// Mitsubishi GX Works2 project: Group22 temp   PLC: FX3G

// global labels: Global1
VAR_GLOBAL
  startMachine AT X010 : BOOL;  (* start machine 1 bottom *)
  machineON AT M0 : BOOL;  (* indication for machine 1 is on *)
  senTouch AT X001 : BOOL;  (* is on if the sensor for the machine sense a tray to execute ziluf *)
  sen_30 AT X003 : BOOL;  (* indication for lower temperature then 30 *)
  sen_15 AT X002 : BOOL;  (* indication for lower temperature then 15 *)
  startDay AT X007 : BOOL;  (* start day bottom *)
  creamInput AT D1119 : REAL;  (* input for cream inventory *)
  creamQuantity AT D1121 : REAL;  (* current quantity of cream in the inventory *)
  chocolateInput AT D1123 : REAL;  (* input for chocolate inventory *)
  chocolateQuantity AT D1125 : REAL;  (* chocolate current quantity *)
  biscuitInput AT D1127 : REAL;  (* input for biscuit inventory *)
  biscuitQuantity AT D1129 : REAL;  (* biscuit current quantity *)
END_VAR
VAR_GLOBAL CONSTANT
  minCream : REAL := 300;  (* minimum quantity needed of cream *)
  minChocolate : REAL := 240;  (* minimum quantity needed of chocolate *)
  minBiscuit : REAL := 6;  (* minimum quantity needed of biscuite *)
END_VAR
VAR_GLOBAL
  notAllQuantitiesGood AT M1 : BOOL;  (* is on if NOT all input quantities are enough for starting the day *)
  counter3sec AT TC1 : BOOL;  (* counter for the y7 blinks at the end of the day *)
END_VAR
VAR_GLOBAL CONSTANT
  fullTime : INT := 30;  (* time of blinking y7 at end day *)
END_VAR
VAR_GLOBAL
  stopAfter3Sec AT TS1 : BOOL;  (* counter for stop blinking of Y7 after 3 seconds *)
  timerReset AT M3 : BOOL;  (* rest timer for counter 5 units packed *)
  timer1 AT TC2 : BOOL;  (* timer name for blinking time of M4 *)
END_VAR
VAR_GLOBAL CONSTANT
  timeInterval : INT := 5;  (* time interval for light on while blinking *)
END_VAR
VAR_GLOBAL
  endTimer1 AT TS2 : BOOL;  (* end timer for blinking fictive light *)
  timer2 AT TC3 : BOOL;  (* timer name for blinking time of M5 *)
  endTimer2 AT TS3 : BOOL;  (* end timer for blinking fictive light that represents Y7 *)
  productionLight AT Y007 : BOOL;  (* light that works all day *)
  fictiveBlinkLight1 AT M4 : BOOL;  (* fictive light that blinks together with Y7 to stimulate Y7 blinks *)
  fictiveBlinkLight2 AT M5 : BOOL;  (* fictive light that represents Y7 *)
  fictiveProductionLight AT M6 : BOOL;  (* production day - process is currently happening *)
  startZilof AT X011 : BOOL;  (* transfer cream from inventory to containter to start zilof stage *)
END_VAR
VAR_GLOBAL CONSTANT
  creamToUse : REAL := 300;  (* amount of cream to use in 1 iteration *)
  biscuitToUse : REAL := 6;  (* amount of bixcuit to use in 1 iteration *)
END_VAR
VAR_GLOBAL
  zilofContainer AT D1131 : REAL;  (* current quantity of cream in the container *)
  counter4seC AT TS4 : BOOL;  (* counter time to blink while transfering *)
END_VAR
VAR_GLOBAL CONSTANT
  blinkTime : INT := 40;  (* time of blinking y0 and y1 at transport from zilof stage to dipping stage *)
END_VAR
VAR_GLOBAL
  timerReset2 AT M7 : BOOL;  (* reset timer for counter of last unit to pack *)
  timer3 AT TC5 : BOOL;  (* timer name for blinking time of Y0 *)
  endTimer3 AT TS5 : BOOL;  (* end timer for blinking Y0 *)
  lightBlink1 AT Y000 : BOOL;  (* blinkig light Y0 to moving units form ziluf *)
  timer4 AT TC6 : BOOL;  (* timer name for blinking time of Y1 *)
  lightBlink2 AT Y001 : BOOL;  (* blinkig light Y1 to moving units form ziluf *)
  endTimer4 AT TS6 : BOOL;  (* end timer for blinking Y1 *)
  zilufON AT Y004 : BOOL;  (* light that stay on while we are in zilof stage *)
  cam AT X004 : BOOL;  (* indication for finish zilof stage *)
  dipInChocolate AT X006 : BOOL;  (* sample the analog input 1 *)
  dipTimer AT TC7 : BOOL;  (* timer for the dipping stage *)
END_VAR
VAR_GLOBAL CONSTANT
  dipInterval : INT := 50;  (* duration time to dip in chocolate *)
END_VAR
VAR_GLOBAL
  dipStop AT TS7 : BOOL;  (* after 5 seconds Y3 sets off *)
  dipInChocolateOn AT Y003 : BOOL;  (* indication for dip process *)
  afterZiluf AT M8 : BOOL;  (* the tray is out of machine a, finished zilufh *)
  iterationDone AT M100 : BOOL;  (* full iteration tray production is done *)
  finishtransferBlink AT M9 : BOOL;  (* after blinking for 4 seconds, turns on *)
  shutDown AT X005 : BOOL;  (* emergency bottom *)
  sampleValue AT D8201 : INT;  (* sample value from anaolog input 1 *)
END_VAR
VAR_GLOBAL CONSTANT
  normalizationFactor : INT := 400;  (* factor to make analog input value shown as the screen *)
END_VAR
VAR_GLOBAL
  finishSampleAnalog AT M10 : BOOL;  (* done sampaling from analog 1 *)
  analog_input_1 AT D8280 : INT;  (* analog input 1 value *)
END_VAR
VAR_GLOBAL CONSTANT
  maxNormalDip : INT := 6;  (* if sample is less than 6 then normal dip *)
END_VAR
VAR_GLOBAL
  normalChocolateDip AT M11 : BOOL;  (* normal chocolate needed *)
  doubledChocolateDip AT M12 : BOOL;  (* double chocolate dip needed *)
END_VAR
VAR_GLOBAL CONSTANT
  amountDoubledDip : REAL := 240;  (* amount of chocolate to coat a tray with doubled amount *)
  amountNormalDip : REAL := 120;  (* amount of chocolate to coat a tray with normal amount *)
END_VAR
VAR_GLOBAL
  coatContainer AT D1135 : REAL;  (* container for coating chocolate above kremboes *)
  finishFillCoatContainer AT M13 : BOOL;  (* indication of end dipping stage *)
  packCounter AT CC1 : BOOL;  (* counter for how much krembo we pack in single iteration *)
END_VAR
VAR_GLOBAL CONSTANT
  packCounterValueLast : INT := 5;  (* number of krembos before the last one *)
END_VAR
VAR_GLOBAL
  packunit AT X000 : BOOL;  (* if on, a krembo unit is getting packed *)
  finishCoating AT M14 : BOOL;  (* if coating process is finished and Y3 turns off *)
  lastPackNeededOn AT Y002 : BOOL;  (* is on if only one last unit left to pack *)
  outCC1 AT CS1 : BOOL;  (* output of counter for 5 unit packs *)
  lastPackCounter AT CC2 : BOOL;  (* counter name of counter for last unit packing *)
END_VAR
VAR_GLOBAL CONSTANT
  packCounterValueLastuUnit : INT := 2;  (* counter for the last unit needed to be packed *)
END_VAR
VAR_GLOBAL
  outCC2 AT CS2 : BOOL;  (* output of counter for last unit pack *)
  readyKrembo AT D2015 : INT;  (* the ready krembos *)
END_VAR
VAR_GLOBAL CONSTANT
  magashKrembo : INT := 6;  (* number of krembos in one iteration *)
END_VAR
VAR_GLOBAL
  kremboOutput AT D8282 : INT;  (* output for the number o ready krembos in tens *)
END_VAR
VAR_GLOBAL CONSTANT
  normalizationFactor2 : INT := 40;  (* factor to make analog input value shown as the screen *)
END_VAR
VAR_GLOBAL
  enoughCreamInContainer AT M15 : BOOL;  (* indication of enough cream in the container to start zilof stage *)
  afterMovingToZilufContainer AT M20 : BOOL;  (* help light to indicate that we are after moving to ziluf container *)
END_VAR

// task Task_01 (event TRUE, interval 0, priority 31): POU_01

PROGRAM POU_01
(* structured ladder/FBD written out as ST: instructions are called as NAME(EN, inputs, outputs); _pN, _eN, _tN stand for wires *)
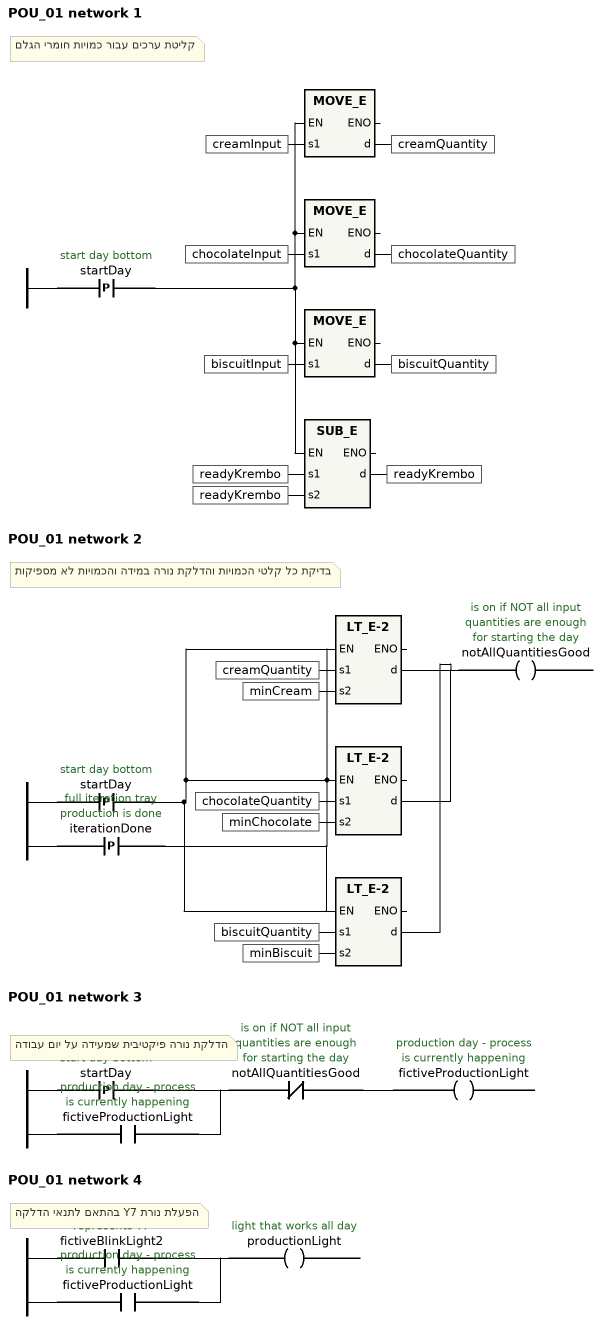
(* network 1 *)
(* קליטת ערכים עבור כמויות חומרי הגלם *)
_p1 := LDP(TRUE, startDay);
MOVE_E(_p1, creamInput, creamQuantity);
MOVE_E(_p1, chocolateInput, chocolateQuantity);
MOVE_E(_p1, biscuitInput, biscuitQuantity);
SUB_E(_p1, readyKrembo, readyKrembo, readyKrembo);
(* network 2 *)
(* בדיקת כל קלטי הכמויות והדלקת נורה במידה והכמויות לא מספיקות *)
_p1 := LDP(TRUE, startDay) OR LDP(TRUE, iterationDone);
LT_E(_p1, creamQuantity, minCream, _t2);
LT_E(_p1, chocolateQuantity, minChocolate, _t3);
LT_E(_p1, biscuitQuantity, minBiscuit, _t4);
notAllQuantitiesGood := _t2 OR _t3 OR _t4;
(* network 3 *)
(* הדלקת נורה פיקטיבית שמעידה על יום עבודה *)
fictiveProductionLight := (LDP(TRUE, startDay) OR fictiveProductionLight) AND NOT notAllQuantitiesGood;
(* network 4 *)
(* הפעלת נורת Y7 בהתאם לתנאי הדלקה *)
productionLight := fictiveBlinkLight2 OR fictiveProductionLight;
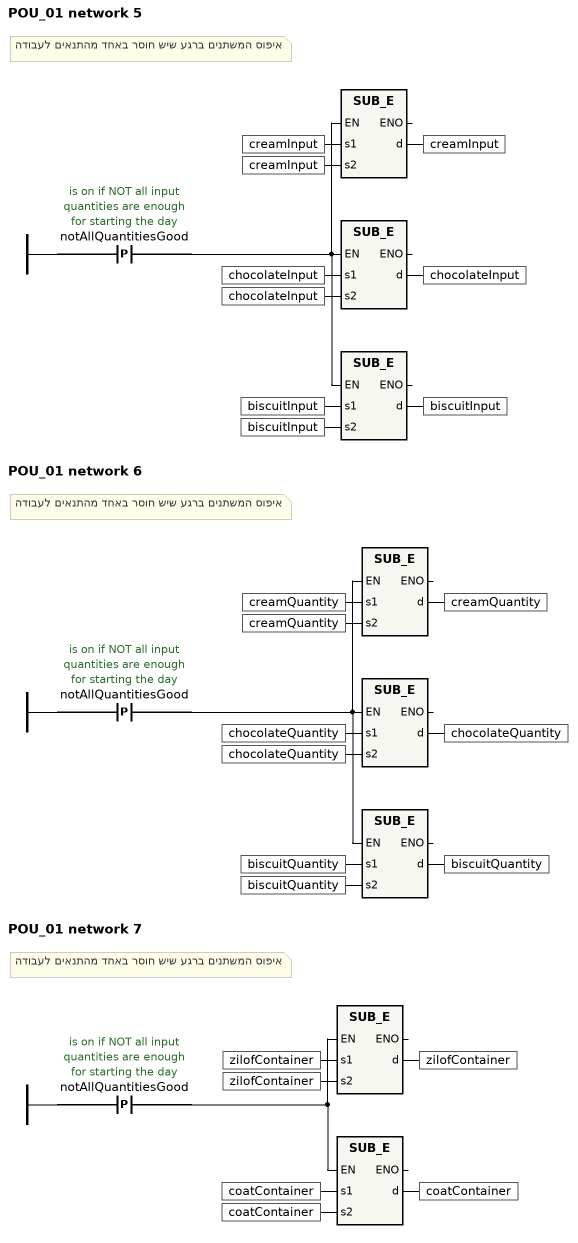
(* network 5 *)
(* איפוס המשתנים ברגע שיש חוסר באחד מהתנאים לעבודה *)
_p1 := LDP(TRUE, notAllQuantitiesGood);
SUB_E(_p1, creamInput, creamInput, creamInput);
SUB_E(_p1, chocolateInput, chocolateInput, chocolateInput);
SUB_E(_p1, biscuitInput, biscuitInput, biscuitInput);
(* network 6 *)
(* איפוס המשתנים ברגע שיש חוסר באחד מהתנאים לעבודה *)
_p1 := LDP(TRUE, notAllQuantitiesGood);
SUB_E(_p1, creamQuantity, creamQuantity, creamQuantity);
SUB_E(_p1, chocolateQuantity, chocolateQuantity, chocolateQuantity);
SUB_E(_p1, biscuitQuantity, biscuitQuantity, biscuitQuantity);
(* network 7 *)
(* איפוס המשתנים ברגע שיש חוסר באחד מהתנאים לעבודה *)
_p1 := LDP(TRUE, notAllQuantitiesGood);
SUB_E(_p1, zilofContainer, zilofContainer, zilofContainer);
SUB_E(_p1, coatContainer, coatContainer, coatContainer);
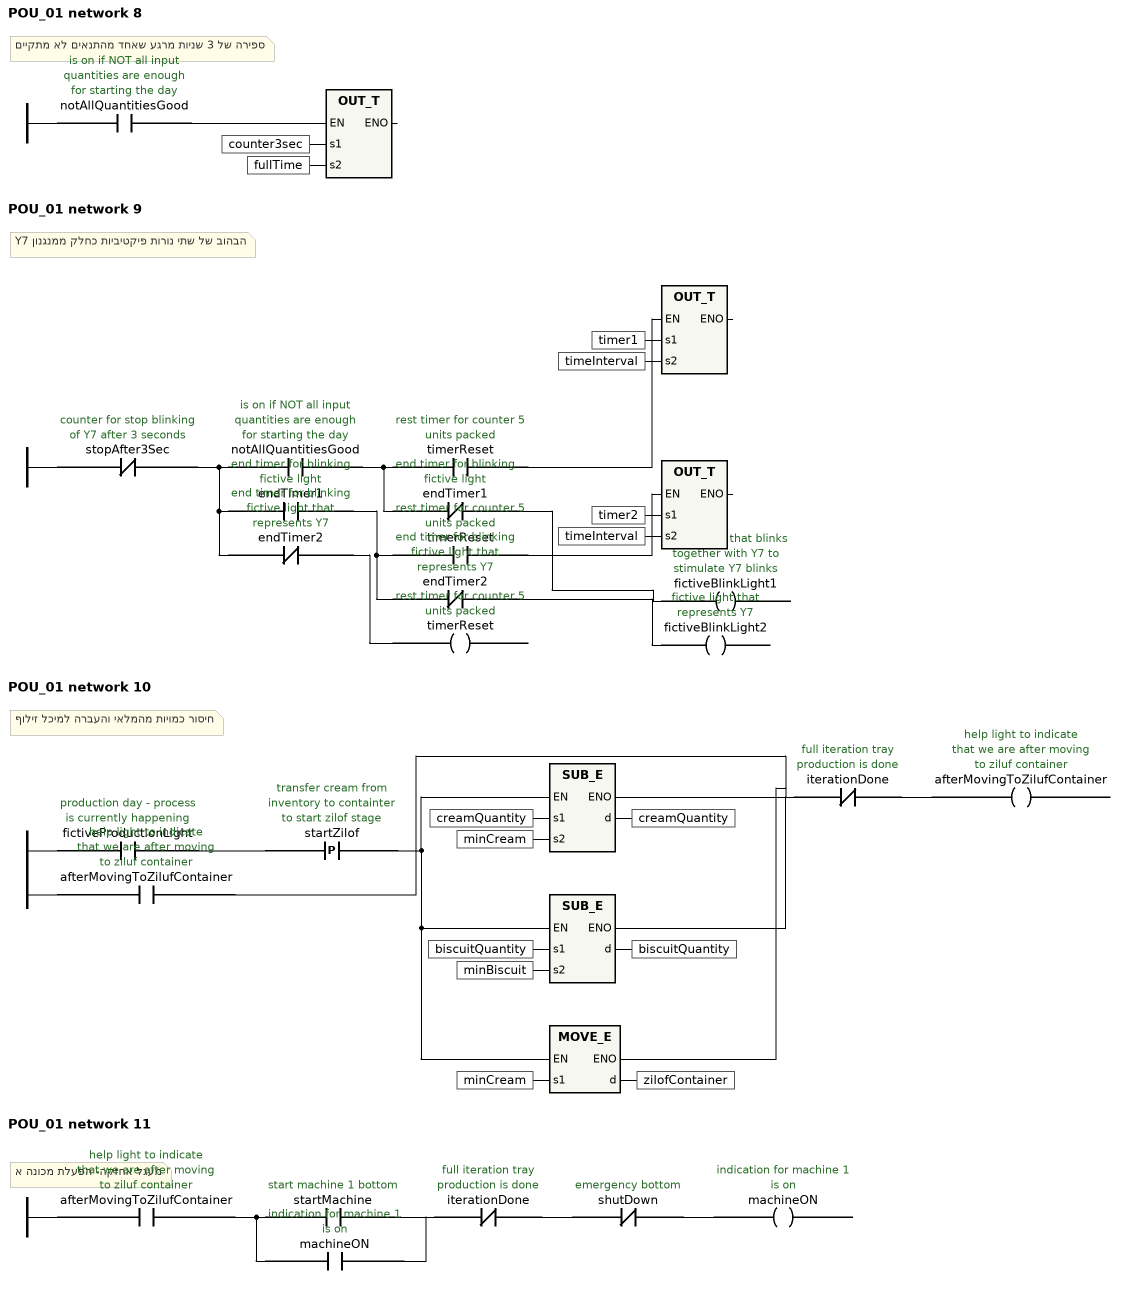
(* network 8 *)
(* ספירה של 3 שניות מרגע שאחד מהתנאים לא מתקיים *)
OUT_T(notAllQuantitiesGood, counter3sec, fullTime);
(* network 9 *)
(* הבהוב של שתי נורות פיקטיביות כחלק ממנגנון Y7 *)
_p1 := NOT stopAfter3Sec;
_p2 := _p1 AND notAllQuantitiesGood;
OUT_T(_p2 AND timerReset, timer1, timeInterval);
fictiveBlinkLight1 := _p2 AND NOT endTimer1;
_p3 := _p1 AND endTimer1;
OUT_T(_p3 AND timerReset, timer2, timeInterval);
fictiveBlinkLight2 := _p3 AND NOT endTimer2;
timerReset := _p1 AND NOT endTimer2;
(* network 10 *)
(* חיסור כמויות מהמלאי והעברה למיכל זילוף *)
_p1 := fictiveProductionLight AND LDP(TRUE, startZilof);
_e2 := SUB_E(_p1, creamQuantity, minCream, creamQuantity);
_e3 := SUB_E(_p1, biscuitQuantity, minBiscuit, biscuitQuantity);
_e4 := MOVE_E(_p1, minCream, zilofContainer);
afterMovingToZilufContainer := (_e2 OR _e3 OR _e4 OR afterMovingToZilufContainer) AND NOT iterationDone;
(* network 11 *)
(* מעגל אחזקה- הפעלת מכונה א *)
machineON := (((afterMovingToZilufContainer AND startMachine) OR (afterMovingToZilufContainer AND machineON)) AND NOT iterationDone) AND NOT shutDown;
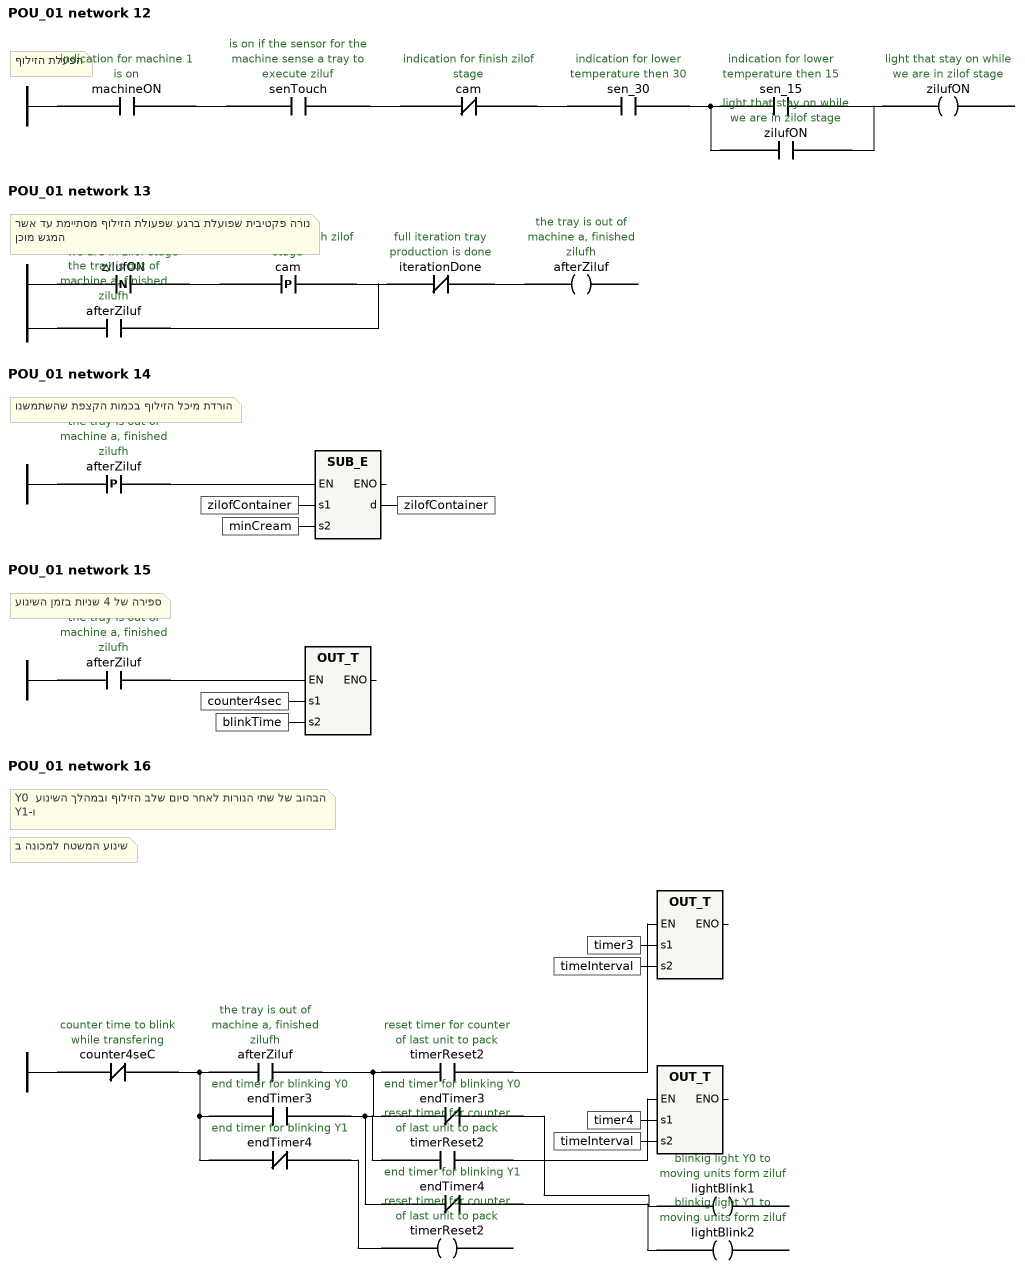
(* network 12 *)
(* הפעלת הזילוף *)
_p1 := machineON AND senTouch AND NOT cam AND sen_30;
zilufON := (_p1 AND sen_15) OR (_p1 AND zilufON);
(* network 13 *)
(* נורה פקטיבית שפועלת ברגע שפעולת הזילוף מסתיימת עד אשר המגש מוכן *)
afterZiluf := ((LDF(TRUE, zilufON) AND LDP(TRUE, cam)) OR afterZiluf) AND NOT iterationDone;
(* network 14 *)
(* הורדת מיכל הזילוף בכמות הקצפת שהשתמשנו *)
SUB_E(LDP(TRUE, afterZiluf), zilofContainer, minCream, zilofContainer);
(* network 15 *)
(* ספירה של 4 שניות בזמן השינוע *)
OUT_T(afterZiluf, counter4sec, blinkTime);
(* network 16 *)
(* הבהוב של שתי הנורות לאחר סיום שלב הזילוף ובמהלך השינוע  Y0 ו-Y1 *)
(* שינוע המשטח למכונה ב *)
_p1 := NOT counter4seC;
_p2 := _p1 AND afterZiluf;
OUT_T(_p2 AND timerReset2, timer3, timeInterval);
lightBlink1 := _p2 AND NOT endTimer3;
_p3 := _p1 AND endTimer3;
OUT_T(_p3 AND timerReset2, timer4, timeInterval);
lightBlink2 := _p3 AND NOT endTimer4;
timerReset2 := _p1 AND NOT endTimer4;
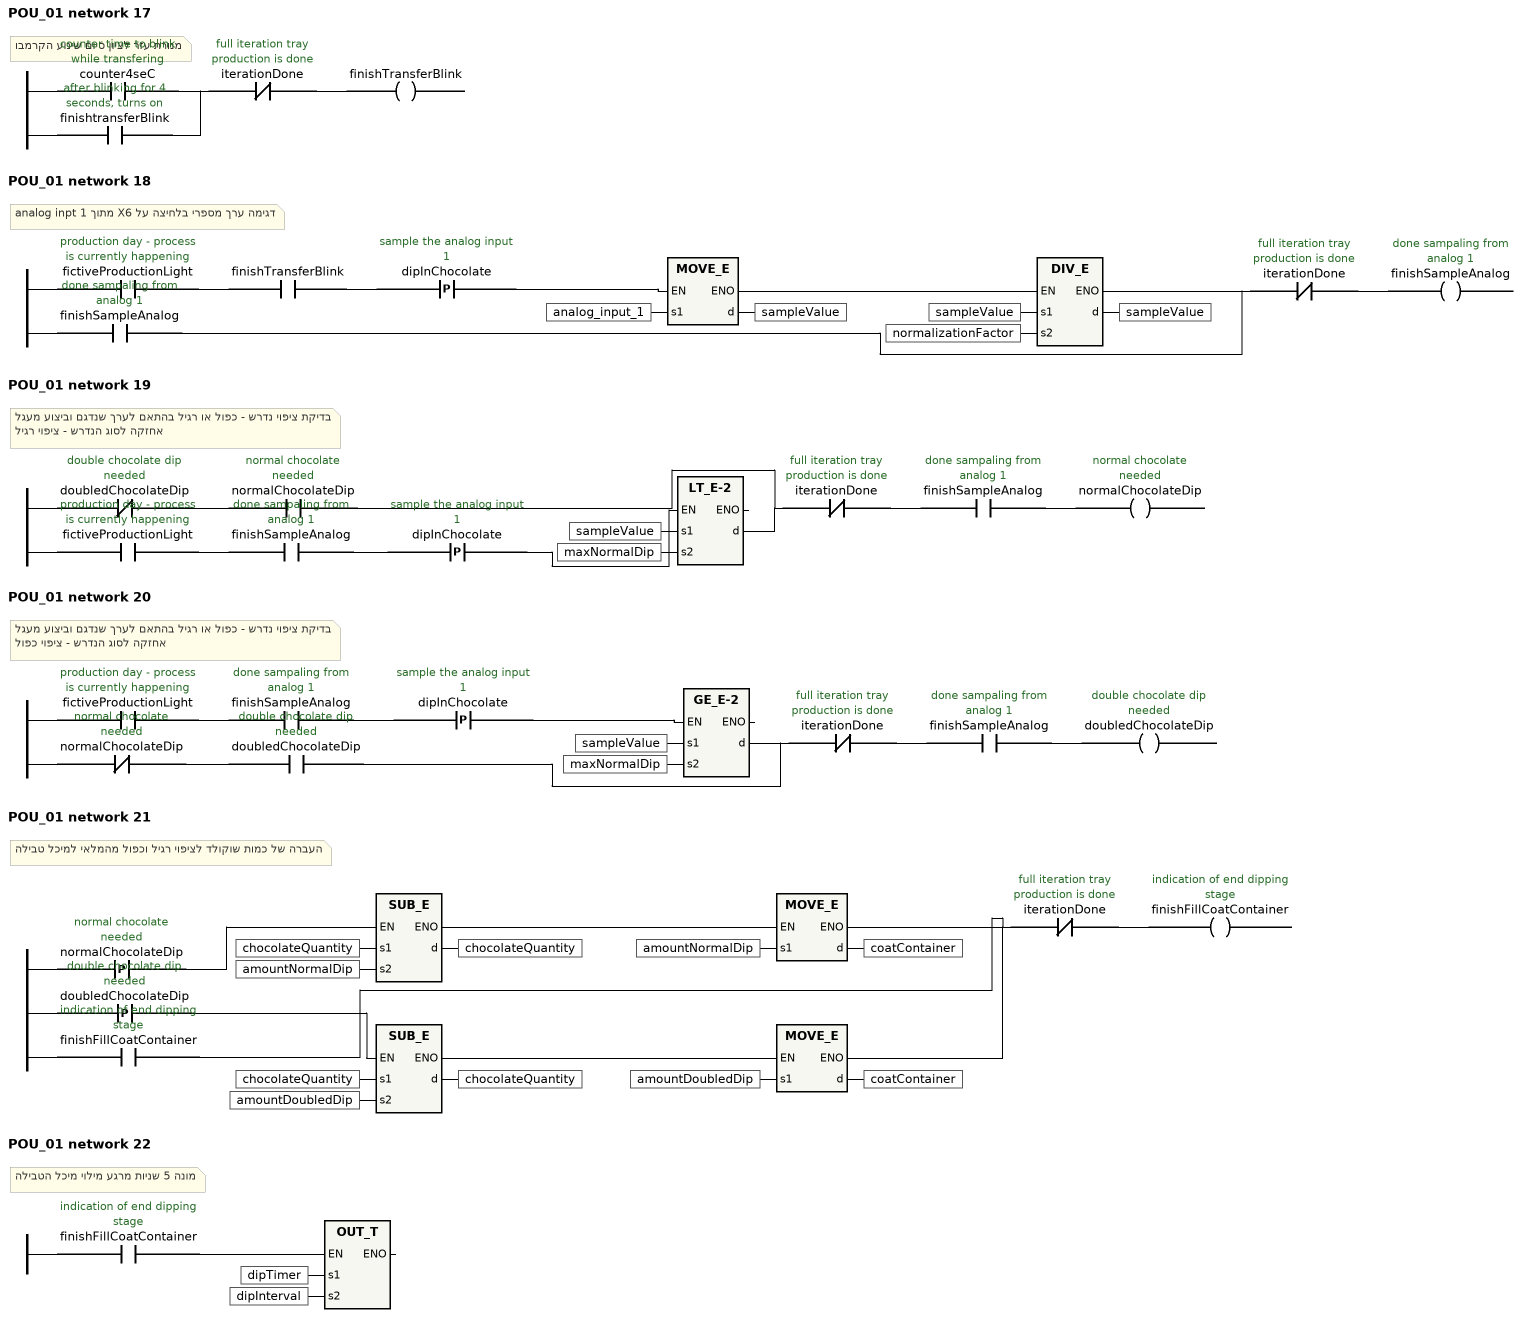
(* network 17 *)
(* מנורת עזר לציון סיום שינוע הקרמבו *)
finishTransferBlink := (counter4seC OR finishtransferBlink) AND NOT iterationDone;
(* network 18 *)
(* דגימה ערך מספרי בלחיצה על X6 מתוך analog inpt 1 *)
_e1 := MOVE_E(fictiveProductionLight AND finishTransferBlink AND LDP(TRUE, dipInChocolate), analog_input_1, sampleValue);
_e2 := DIV_E(_e1, sampleValue, normalizationFactor, sampleValue);
finishSampleAnalog := (_e2 OR finishSampleAnalog) AND NOT iterationDone;
(* network 19 *)
(* בדיקת ציפוי נדרש - כפול או רגיל בהתאם לערך שנדגם וביצוע מעגל אחזקה לסוג הנדרש - ציפוי רגיל *)
LT_E(fictiveProductionLight AND finishSampleAnalog AND LDP(TRUE, dipInChocolate), sampleValue, maxNormalDip, _t1);
normalChocolateDip := (((NOT doubledChocolateDip AND normalChocolateDip) OR _t1) AND NOT iterationDone) AND finishSampleAnalog;
(* network 20 *)
(* בדיקת ציפוי נדרש - כפול או רגיל בהתאם לערך שנדגם וביצוע מעגל אחזקה לסוג הנדרש - ציפוי כפול *)
GE_E(fictiveProductionLight AND finishSampleAnalog AND LDP(TRUE, dipInChocolate), sampleValue, maxNormalDip, _t1);
doubledChocolateDip := ((_t1 OR (NOT normalChocolateDip AND doubledChocolateDip)) AND NOT iterationDone) AND finishSampleAnalog;
(* network 21 *)
(* העברה של כמות שוקולד לציפוי רגיל וכפול מהמלאי למיכל טבילה *)
_e1 := SUB_E(LDP(TRUE, normalChocolateDip), chocolateQuantity, amountNormalDip, chocolateQuantity);
_e2 := MOVE_E(_e1, amountNormalDip, coatContainer);
_e3 := SUB_E(LDP(TRUE, doubledChocolateDip), chocolateQuantity, amountDoubledDip, chocolateQuantity);
_e4 := MOVE_E(_e3, amountDoubledDip, coatContainer);
finishFillCoatContainer := (_e2 OR _e4 OR finishFillCoatContainer) AND NOT iterationDone;
(* network 22 *)
(* מונה 5 שניות מרגע מילוי מיכל הטבילה *)
OUT_T(finishFillCoatContainer, dipTimer, dipInterval);
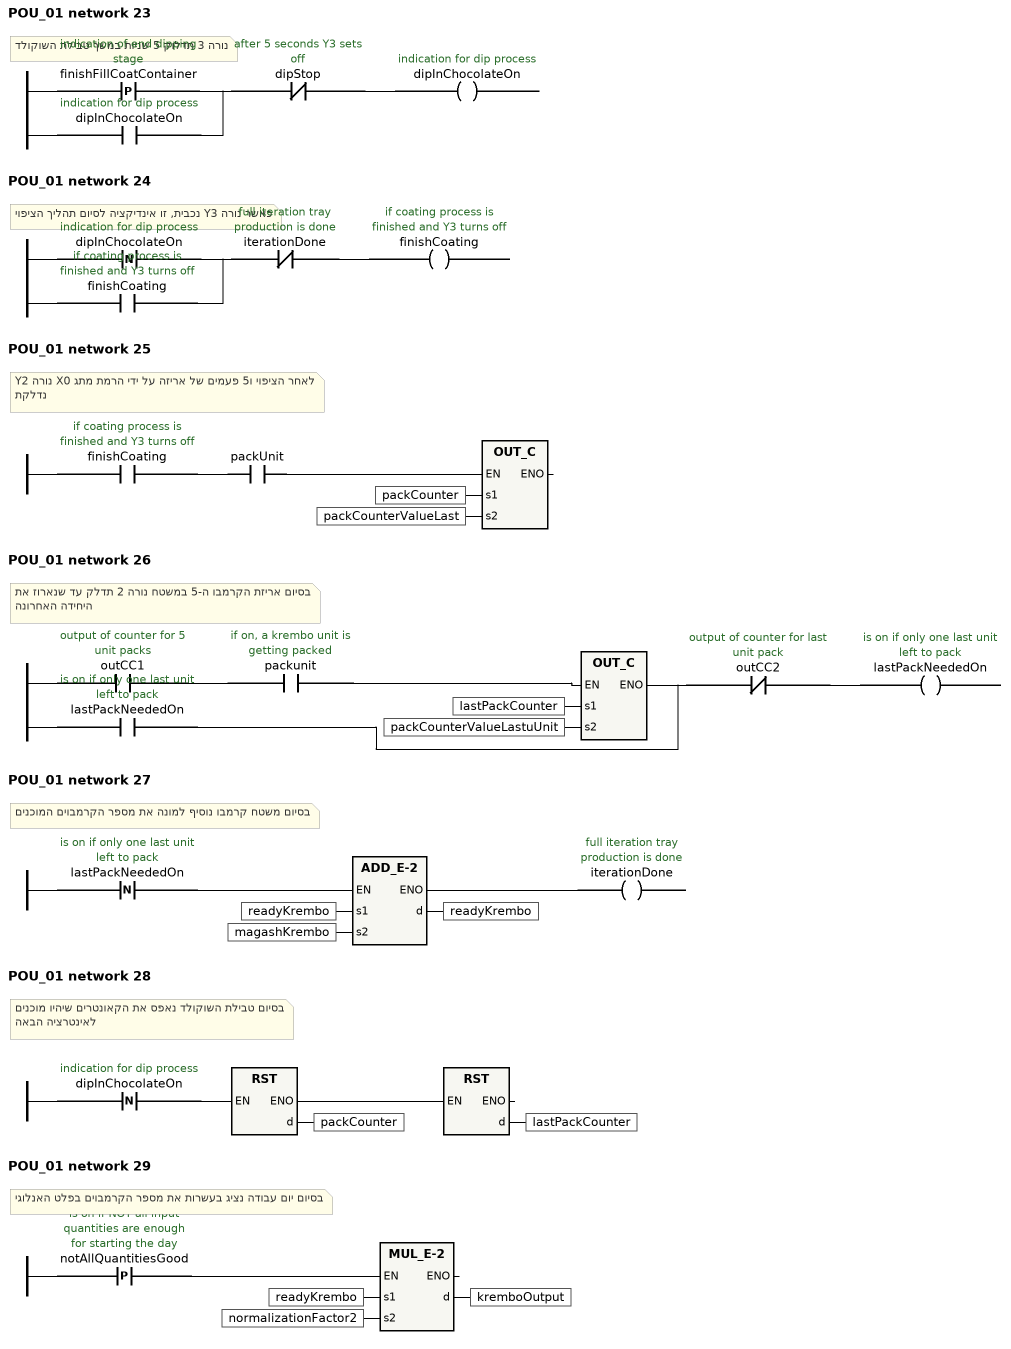
(* network 23 *)
(* נורה 3 תדלוק 5 שניות במשך טבילת השוקולד *)
dipInChocolateOn := (LDP(TRUE, finishFillCoatContainer) OR dipInChocolateOn) AND NOT dipStop;
(* network 24 *)
(* כאשר נורה Y3 נכבית, זו אינדיקציה לסיום תהליך הציפוי *)
finishCoating := (LDF(TRUE, dipInChocolateOn) OR finishCoating) AND NOT iterationDone;
(* network 25 *)
(* לאחר הציפוי ו5 פעמים של אריזה על ידי הרמת מתג X0 נורה Y2 נדלקת *)
OUT_C(finishCoating AND packUnit, packCounter, packCounterValueLast);
(* network 26 *)
(* בסיום אריזת הקרמבו ה-5 במשטח נורה 2 תדלק עד שנארוז את היחידה האחרונה *)
_e1 := OUT_C(outCC1 AND packunit, lastPackCounter, packCounterValueLastuUnit);
lastPackNeededOn := (_e1 OR lastPackNeededOn) AND NOT outCC2;
(* network 27 *)
(* בסיום משטח קרמבו נוסיף למונה את מספר הקרמבוים המוכנים *)
_e1 := ADD_E(LDF(TRUE, lastPackNeededOn), readyKrembo, magashKrembo, readyKrembo);
iterationDone := _e1;
(* network 28 *)
(* בסיום טבילת השוקולד נאפס את הקאונטרים שיהיו מוכנים לאינטרציה הבאה *)
_e1 := RST(LDF(TRUE, dipInChocolateOn), packCounter);
RST(_e1, lastPackCounter);
(* network 29 *)
(* בסיום יום עבודה נציג בעשרות את מספר הקרמבוים בפלט האנלוגי *)
MUL_E(LDP(TRUE, notAllQuantitiesGood), readyKrembo, normalizationFactor2, kremboOutput);
END_PROGRAM
